(* CODESYS project IndraLogic.project

Project tree, tasks and I/O mapping:
  IndraMotionMlc1 : IndraMotion MLC L25, Bosch Rexroth AG, order no. R911171363, version 14.20.34.0
    application Application
      libraries: VisuDialogs, * (System)
      task PlcTask (cyclic, interval 25 ms, priority 5, watchdog 100 ms x 2) calls prgVisualization, prgDataSimulator, PrgBedinpult_Visu
      global variables UserVarGlobal
      Symbols
      global variables MlcVarGlobal
      image pool ImagePool
      Funktionsbausteine/
        function block GenAngleTest [ST]
        function block GenNumTest [ST]
        function block TestGen [FBD]
        function block Tweener [SFC]: SetResToStart, IncResult, DecResult, SetResultToFinal
      Programme/
        program prgVisualization [ST]
        program prgDataSimulator [ST]
      Structs/
        data type TestStruct
      Bedinpult_Visu/
        program PrgBedinpult_Visu [LD]
      HMI/
        visualisation viAttitudeIndicator
      Frames/
        visualisation frBedinpult
        visualisation frSelfTestLamp
    Inline_I_O : Inline I/O, Bosch Rexroth AG, version 12.8.2.0
    Sercos_III_Master : SercosIII Master, Rexroth, order no. 1, version 14.6.0.0
  text list GlobalTextList
  5ce3da45-db07-42e7-a21c-a00fff4ed8f6|C:\Users\Kun\Desktop\Uni\Automatisierungstechnik\ProjektaufgabeAT\Overlay.png
  5ce3da45-db07-42e7-a21c-a00fff4ed8f6|C:\Users\Ghaith\Desktop\Modellfabrik\Logo.jpg
*)

// IndraMotionMlc1/Application/Structs/TestStruct
TYPE TestStruct :
STRUCT
	bEnable		: BOOL;
	iStartValue	: INT;
	iFinalValue	: INT;
	rSweepInc	: REAL;
	bTestActive	: BOOL;
END_STRUCT
END_TYPE

// IndraMotionMlc1/Application/UserVarGlobal
{attribute 'qualified_only'}
VAR_GLOBAL
	bSelfTestAtStartup : BOOL	:= TRUE;
	
	rPitch 		: 	REAL;
	rRoll 		: 	REAL;
	iHeight		:	INT;
	uiSpeed		:	UINT;
	
	rPitch_Input 		: 	REAL;
	rRoll_Input 		: 	REAL;
	iHeight_Input		:	INT;
	uiSpeed_Input		:	UINT;
	
	bAutomatic_Mode_Input	: BOOL;
END_VAR

// IndraMotionMlc1/Application/MlcVarGlobal
(* Automatically generated code by XLC/MLC. *)
(* Please don't edit, the code will be overwritten. For usercode use UserVarGlobal! *)
{attribute 'linkalways'}
{attribute 'analysis' := '-33'}
VAR_GLOBAL CONSTANT

(*Probe 001*)
TouchProbe001: TOUCHPROBE_REF :=(CntrlNo:=LOCAL_CNTRL,TouchProbeNo:=TOUCHPROBE_1);

(*Probe 002*)
TouchProbe002: TOUCHPROBE_REF :=(CntrlNo:=LOCAL_CNTRL,TouchProbeNo:=TOUCHPROBE_2);

(*Probe 003*)
TouchProbe003: TOUCHPROBE_REF :=(CntrlNo:=LOCAL_CNTRL,TouchProbeNo:=TOUCHPROBE_3);

(*Probe 004*)
TouchProbe004: TOUCHPROBE_REF :=(CntrlNo:=LOCAL_CNTRL,TouchProbeNo:=TOUCHPROBE_4);

(*Probe 005*)
TouchProbe005: TOUCHPROBE_REF :=(CntrlNo:=LOCAL_CNTRL,TouchProbeNo:=TOUCHPROBE_5);

(*Probe 006*)
TouchProbe006: TOUCHPROBE_REF :=(CntrlNo:=LOCAL_CNTRL,TouchProbeNo:=TOUCHPROBE_6);

(*Probe 007*)
TouchProbe007: TOUCHPROBE_REF :=(CntrlNo:=LOCAL_CNTRL,TouchProbeNo:=TOUCHPROBE_7);

(*Probe 008*)
TouchProbe008: TOUCHPROBE_REF :=(CntrlNo:=LOCAL_CNTRL,TouchProbeNo:=TOUCHPROBE_8);

(*Probe 009*)
TouchProbe009: TOUCHPROBE_REF :=(CntrlNo:=LOCAL_CNTRL,TouchProbeNo:=TOUCHPROBE_9);

(*Probe 010*)
TouchProbe010: TOUCHPROBE_REF :=(CntrlNo:=LOCAL_CNTRL,TouchProbeNo:=TOUCHPROBE_10);

(*Probe 011*)
TouchProbe011: TOUCHPROBE_REF :=(CntrlNo:=LOCAL_CNTRL,TouchProbeNo:=TOUCHPROBE_11);

(*Probe 012*)
TouchProbe012: TOUCHPROBE_REF :=(CntrlNo:=LOCAL_CNTRL,TouchProbeNo:=TOUCHPROBE_12);

(*Probe 013*)
TouchProbe013: TOUCHPROBE_REF :=(CntrlNo:=LOCAL_CNTRL,TouchProbeNo:=TOUCHPROBE_13);

(*Probe 014*)
TouchProbe014: TOUCHPROBE_REF :=(CntrlNo:=LOCAL_CNTRL,TouchProbeNo:=TOUCHPROBE_14);

(*Probe 015*)
TouchProbe015: TOUCHPROBE_REF :=(CntrlNo:=LOCAL_CNTRL,TouchProbeNo:=TOUCHPROBE_15);

(*Probe 016*)
TouchProbe016: TOUCHPROBE_REF :=(CntrlNo:=LOCAL_CNTRL,TouchProbeNo:=TOUCHPROBE_16);

(*Probe 017*)
TouchProbe017: TOUCHPROBE_REF :=(CntrlNo:=LOCAL_CNTRL,TouchProbeNo:=TOUCHPROBE_17);

(*Probe 018*)
TouchProbe018: TOUCHPROBE_REF :=(CntrlNo:=LOCAL_CNTRL,TouchProbeNo:=TOUCHPROBE_18);

(*Probe 019*)
TouchProbe019: TOUCHPROBE_REF :=(CntrlNo:=LOCAL_CNTRL,TouchProbeNo:=TOUCHPROBE_19);

(*Probe 020*)
TouchProbe020: TOUCHPROBE_REF :=(CntrlNo:=LOCAL_CNTRL,TouchProbeNo:=TOUCHPROBE_20);

(*Probe 021*)
TouchProbe021: TOUCHPROBE_REF :=(CntrlNo:=LOCAL_CNTRL,TouchProbeNo:=TOUCHPROBE_21);

(*Probe 022*)
TouchProbe022: TOUCHPROBE_REF :=(CntrlNo:=LOCAL_CNTRL,TouchProbeNo:=TOUCHPROBE_22);

(*Probe 023*)
TouchProbe023: TOUCHPROBE_REF :=(CntrlNo:=LOCAL_CNTRL,TouchProbeNo:=TOUCHPROBE_23);

(*Probe 024*)
TouchProbe024: TOUCHPROBE_REF :=(CntrlNo:=LOCAL_CNTRL,TouchProbeNo:=TOUCHPROBE_24);

(*Probe 025*)
TouchProbe025: TOUCHPROBE_REF :=(CntrlNo:=LOCAL_CNTRL,TouchProbeNo:=TOUCHPROBE_25);

(*Probe 026*)
TouchProbe026: TOUCHPROBE_REF :=(CntrlNo:=LOCAL_CNTRL,TouchProbeNo:=TOUCHPROBE_26);

(*Probe 027*)
TouchProbe027: TOUCHPROBE_REF :=(CntrlNo:=LOCAL_CNTRL,TouchProbeNo:=TOUCHPROBE_27);

(*Probe 028*)
TouchProbe028: TOUCHPROBE_REF :=(CntrlNo:=LOCAL_CNTRL,TouchProbeNo:=TOUCHPROBE_28);

(*Probe 029*)
TouchProbe029: TOUCHPROBE_REF :=(CntrlNo:=LOCAL_CNTRL,TouchProbeNo:=TOUCHPROBE_29);

(*Probe 030*)
TouchProbe030: TOUCHPROBE_REF :=(CntrlNo:=LOCAL_CNTRL,TouchProbeNo:=TOUCHPROBE_30);

(*Probe 031*)
TouchProbe031: TOUCHPROBE_REF :=(CntrlNo:=LOCAL_CNTRL,TouchProbeNo:=TOUCHPROBE_31);

(*Probe 032*)
TouchProbe032: TOUCHPROBE_REF :=(CntrlNo:=LOCAL_CNTRL,TouchProbeNo:=TOUCHPROBE_32);

(*Probe 033*)
TouchProbe033: TOUCHPROBE_REF :=(CntrlNo:=LOCAL_CNTRL,TouchProbeNo:=TOUCHPROBE_33);

(*Probe 034*)
TouchProbe034: TOUCHPROBE_REF :=(CntrlNo:=LOCAL_CNTRL,TouchProbeNo:=TOUCHPROBE_34);

(*Probe 035*)
TouchProbe035: TOUCHPROBE_REF :=(CntrlNo:=LOCAL_CNTRL,TouchProbeNo:=TOUCHPROBE_35);

(*Probe 036*)
TouchProbe036: TOUCHPROBE_REF :=(CntrlNo:=LOCAL_CNTRL,TouchProbeNo:=TOUCHPROBE_36);

(*Probe 037*)
TouchProbe037: TOUCHPROBE_REF :=(CntrlNo:=LOCAL_CNTRL,TouchProbeNo:=TOUCHPROBE_37);

(*Probe 038*)
TouchProbe038: TOUCHPROBE_REF :=(CntrlNo:=LOCAL_CNTRL,TouchProbeNo:=TOUCHPROBE_38);

(*Probe 039*)
TouchProbe039: TOUCHPROBE_REF :=(CntrlNo:=LOCAL_CNTRL,TouchProbeNo:=TOUCHPROBE_39);

(*Probe 040*)
TouchProbe040: TOUCHPROBE_REF :=(CntrlNo:=LOCAL_CNTRL,TouchProbeNo:=TOUCHPROBE_40);

(*Probe 041*)
TouchProbe041: TOUCHPROBE_REF :=(CntrlNo:=LOCAL_CNTRL,TouchProbeNo:=TOUCHPROBE_41);

(*Probe 042*)
TouchProbe042: TOUCHPROBE_REF :=(CntrlNo:=LOCAL_CNTRL,TouchProbeNo:=TOUCHPROBE_42);

(*Probe 043*)
TouchProbe043: TOUCHPROBE_REF :=(CntrlNo:=LOCAL_CNTRL,TouchProbeNo:=TOUCHPROBE_43);

(*Probe 044*)
TouchProbe044: TOUCHPROBE_REF :=(CntrlNo:=LOCAL_CNTRL,TouchProbeNo:=TOUCHPROBE_44);

(*Probe 045*)
TouchProbe045: TOUCHPROBE_REF :=(CntrlNo:=LOCAL_CNTRL,TouchProbeNo:=TOUCHPROBE_45);

(*Probe 046*)
TouchProbe046: TOUCHPROBE_REF :=(CntrlNo:=LOCAL_CNTRL,TouchProbeNo:=TOUCHPROBE_46);

(*Probe 047*)
TouchProbe047: TOUCHPROBE_REF :=(CntrlNo:=LOCAL_CNTRL,TouchProbeNo:=TOUCHPROBE_47);

(*Probe 048*)
TouchProbe048: TOUCHPROBE_REF :=(CntrlNo:=LOCAL_CNTRL,TouchProbeNo:=TOUCHPROBE_48);

(*Probe 049*)
TouchProbe049: TOUCHPROBE_REF :=(CntrlNo:=LOCAL_CNTRL,TouchProbeNo:=TOUCHPROBE_49);

(*Probe 050*)
TouchProbe050: TOUCHPROBE_REF :=(CntrlNo:=LOCAL_CNTRL,TouchProbeNo:=TOUCHPROBE_50);

(*Probe 051*)
TouchProbe051: TOUCHPROBE_REF :=(CntrlNo:=LOCAL_CNTRL,TouchProbeNo:=TOUCHPROBE_51);

(*Probe 052*)
TouchProbe052: TOUCHPROBE_REF :=(CntrlNo:=LOCAL_CNTRL,TouchProbeNo:=TOUCHPROBE_52);

(*Probe 053*)
TouchProbe053: TOUCHPROBE_REF :=(CntrlNo:=LOCAL_CNTRL,TouchProbeNo:=TOUCHPROBE_53);

(*Probe 054*)
TouchProbe054: TOUCHPROBE_REF :=(CntrlNo:=LOCAL_CNTRL,TouchProbeNo:=TOUCHPROBE_54);

(*Probe 055*)
TouchProbe055: TOUCHPROBE_REF :=(CntrlNo:=LOCAL_CNTRL,TouchProbeNo:=TOUCHPROBE_55);

(*Probe 056*)
TouchProbe056: TOUCHPROBE_REF :=(CntrlNo:=LOCAL_CNTRL,TouchProbeNo:=TOUCHPROBE_56);

(*Probe 057*)
TouchProbe057: TOUCHPROBE_REF :=(CntrlNo:=LOCAL_CNTRL,TouchProbeNo:=TOUCHPROBE_57);

(*Probe 058*)
TouchProbe058: TOUCHPROBE_REF :=(CntrlNo:=LOCAL_CNTRL,TouchProbeNo:=TOUCHPROBE_58);

(*Probe 059*)
TouchProbe059: TOUCHPROBE_REF :=(CntrlNo:=LOCAL_CNTRL,TouchProbeNo:=TOUCHPROBE_59);

(*Probe 060*)
TouchProbe060: TOUCHPROBE_REF :=(CntrlNo:=LOCAL_CNTRL,TouchProbeNo:=TOUCHPROBE_60);

(*Probe 061*)
TouchProbe061: TOUCHPROBE_REF :=(CntrlNo:=LOCAL_CNTRL,TouchProbeNo:=TOUCHPROBE_61);

(*Probe 062*)
TouchProbe062: TOUCHPROBE_REF :=(CntrlNo:=LOCAL_CNTRL,TouchProbeNo:=TOUCHPROBE_62);

(*Probe 063*)
TouchProbe063: TOUCHPROBE_REF :=(CntrlNo:=LOCAL_CNTRL,TouchProbeNo:=TOUCHPROBE_63);

(*Probe 064*)
TouchProbe064: TOUCHPROBE_REF :=(CntrlNo:=LOCAL_CNTRL,TouchProbeNo:=TOUCHPROBE_64);

(*Probe 065*)
TouchProbe065: TOUCHPROBE_REF :=(CntrlNo:=LOCAL_CNTRL,TouchProbeNo:=TOUCHPROBE_65);

(*Probe 066*)
TouchProbe066: TOUCHPROBE_REF :=(CntrlNo:=LOCAL_CNTRL,TouchProbeNo:=TOUCHPROBE_66);

(*Probe 067*)
TouchProbe067: TOUCHPROBE_REF :=(CntrlNo:=LOCAL_CNTRL,TouchProbeNo:=TOUCHPROBE_67);

(*Probe 068*)
TouchProbe068: TOUCHPROBE_REF :=(CntrlNo:=LOCAL_CNTRL,TouchProbeNo:=TOUCHPROBE_68);

(*Probe 069*)
TouchProbe069: TOUCHPROBE_REF :=(CntrlNo:=LOCAL_CNTRL,TouchProbeNo:=TOUCHPROBE_69);

(*Probe 070*)
TouchProbe070: TOUCHPROBE_REF :=(CntrlNo:=LOCAL_CNTRL,TouchProbeNo:=TOUCHPROBE_70);

(*Probe 071*)
TouchProbe071: TOUCHPROBE_REF :=(CntrlNo:=LOCAL_CNTRL,TouchProbeNo:=TOUCHPROBE_71);

(*Probe 072*)
TouchProbe072: TOUCHPROBE_REF :=(CntrlNo:=LOCAL_CNTRL,TouchProbeNo:=TOUCHPROBE_72);

(*Probe 073*)
TouchProbe073: TOUCHPROBE_REF :=(CntrlNo:=LOCAL_CNTRL,TouchProbeNo:=TOUCHPROBE_73);

(*Probe 074*)
TouchProbe074: TOUCHPROBE_REF :=(CntrlNo:=LOCAL_CNTRL,TouchProbeNo:=TOUCHPROBE_74);

(*Probe 075*)
TouchProbe075: TOUCHPROBE_REF :=(CntrlNo:=LOCAL_CNTRL,TouchProbeNo:=TOUCHPROBE_75);

(*Probe 076*)
TouchProbe076: TOUCHPROBE_REF :=(CntrlNo:=LOCAL_CNTRL,TouchProbeNo:=TOUCHPROBE_76);

(*Probe 077*)
TouchProbe077: TOUCHPROBE_REF :=(CntrlNo:=LOCAL_CNTRL,TouchProbeNo:=TOUCHPROBE_77);

(*Probe 078*)
TouchProbe078: TOUCHPROBE_REF :=(CntrlNo:=LOCAL_CNTRL,TouchProbeNo:=TOUCHPROBE_78);

(*Probe 079*)
TouchProbe079: TOUCHPROBE_REF :=(CntrlNo:=LOCAL_CNTRL,TouchProbeNo:=TOUCHPROBE_79);

(*Probe 080*)
TouchProbe080: TOUCHPROBE_REF :=(CntrlNo:=LOCAL_CNTRL,TouchProbeNo:=TOUCHPROBE_80);

(*Probe 081*)
TouchProbe081: TOUCHPROBE_REF :=(CntrlNo:=LOCAL_CNTRL,TouchProbeNo:=TOUCHPROBE_81);

(*Probe 082*)
TouchProbe082: TOUCHPROBE_REF :=(CntrlNo:=LOCAL_CNTRL,TouchProbeNo:=TOUCHPROBE_82);

(*Probe 083*)
TouchProbe083: TOUCHPROBE_REF :=(CntrlNo:=LOCAL_CNTRL,TouchProbeNo:=TOUCHPROBE_83);

(*Probe 084*)
TouchProbe084: TOUCHPROBE_REF :=(CntrlNo:=LOCAL_CNTRL,TouchProbeNo:=TOUCHPROBE_84);

(*Probe 085*)
TouchProbe085: TOUCHPROBE_REF :=(CntrlNo:=LOCAL_CNTRL,TouchProbeNo:=TOUCHPROBE_85);

(*Probe 086*)
TouchProbe086: TOUCHPROBE_REF :=(CntrlNo:=LOCAL_CNTRL,TouchProbeNo:=TOUCHPROBE_86);

(*Probe 087*)
TouchProbe087: TOUCHPROBE_REF :=(CntrlNo:=LOCAL_CNTRL,TouchProbeNo:=TOUCHPROBE_87);

(*Probe 088*)
TouchProbe088: TOUCHPROBE_REF :=(CntrlNo:=LOCAL_CNTRL,TouchProbeNo:=TOUCHPROBE_88);

(*Probe 089*)
TouchProbe089: TOUCHPROBE_REF :=(CntrlNo:=LOCAL_CNTRL,TouchProbeNo:=TOUCHPROBE_89);

(*Probe 090*)
TouchProbe090: TOUCHPROBE_REF :=(CntrlNo:=LOCAL_CNTRL,TouchProbeNo:=TOUCHPROBE_90);

(*Probe 091*)
TouchProbe091: TOUCHPROBE_REF :=(CntrlNo:=LOCAL_CNTRL,TouchProbeNo:=TOUCHPROBE_91);

(*Probe 092*)
TouchProbe092: TOUCHPROBE_REF :=(CntrlNo:=LOCAL_CNTRL,TouchProbeNo:=TOUCHPROBE_92);

(*Probe 093*)
TouchProbe093: TOUCHPROBE_REF :=(CntrlNo:=LOCAL_CNTRL,TouchProbeNo:=TOUCHPROBE_93);

(*Probe 094*)
TouchProbe094: TOUCHPROBE_REF :=(CntrlNo:=LOCAL_CNTRL,TouchProbeNo:=TOUCHPROBE_94);

(*Probe 095*)
TouchProbe095: TOUCHPROBE_REF :=(CntrlNo:=LOCAL_CNTRL,TouchProbeNo:=TOUCHPROBE_95);

(*Probe 096*)
TouchProbe096: TOUCHPROBE_REF :=(CntrlNo:=LOCAL_CNTRL,TouchProbeNo:=TOUCHPROBE_96);

(*Probe 097*)
TouchProbe097: TOUCHPROBE_REF :=(CntrlNo:=LOCAL_CNTRL,TouchProbeNo:=TOUCHPROBE_97);

(*Probe 098*)
TouchProbe098: TOUCHPROBE_REF :=(CntrlNo:=LOCAL_CNTRL,TouchProbeNo:=TOUCHPROBE_98);

(*Probe 099*)
TouchProbe099: TOUCHPROBE_REF :=(CntrlNo:=LOCAL_CNTRL,TouchProbeNo:=TOUCHPROBE_99);

(*Probe 100*)
TouchProbe100: TOUCHPROBE_REF :=(CntrlNo:=LOCAL_CNTRL,TouchProbeNo:=TOUCHPROBE_100);

END_VAR

// IndraMotionMlc1/Application/Programme/prgVisualization
PROGRAM prgVisualization
VAR
	rPitch_Visu 	: 	REAL;
	rRoll_Visu		: 	REAL;
	iHeight_Visu		:	INT;
	uiSpeed_Visu		:	UINT;
	bDisableControlPanel: BOOL;
END_VAR

VAR CONSTANT
	
END_VAR

rRoll_Visu := UserVarGlobal.rRoll;
iHeight_Visu := UserVarGlobal.iHeight;
rPitch_Visu := UserVarGlobal.rPitch * 4;
uiSpeed_Visu :=UserVarGlobal.uiSpeed;

IF ((UserVarGlobal.bAutomatic_Mode_Input = FALSE AND (rRoll_Visu <> UserVarGlobal.rRoll_Input OR rPitch_Visu <> UserVarGlobal.rPitch_Input*4 OR iHeight_Visu <> UserVarGlobal.iHeight_Input OR uiSpeed_Visu <> UserVarGlobal.uiSpeed_Input)) OR UserVarGlobal.bSelfTestAtStartup) THEN
	bDisableControlPanel := TRUE;
ELSE
	bDisableControlPanel := FALSE;
END_IF

END_PROGRAM

// IndraMotionMlc1/Application/Programme/prgDataSimulator
PROGRAM prgDataSimulator
VAR
	rPitch 			: 	REAL;
	rRoll 			: 	REAL;
	iHeight			:	INT;
	uiSpeed			:	UINT;
	
	// Internal Variables for Automatic Operation
	fbTestGenerator		:	TestGen;
	suPitchTestStruct	:	testStruct;
	suRollTestStruct	:	testStruct;
	suHeightTestStruct  :	testStruct;
	suSpeedTestStruct	:	testStruct;
	bInit				:	BOOL := TRUE;
	
	// Internal Variables for Manual Operation
	fbPitchTween		: Tweener;
	fbRollTween			: Tweener;
	fbHeightTween		: Tweener;
	fbSpeedTween		: Tweener;
	
	siSweepInc		:	SINT	:=	1;
END_VAR

// Initialize Test Structs
IF bInit THEN
	suRollTestStruct.bEnable 		:= TRUE;
	suRollTestStruct.iStartValue 	:= -30;
	suRollTestStruct.iFinalValue 	:= 30;
	suRollTestStruct.rSweepInc 	:= 0.6;
	
	suHeightTestStruct.bEnable 	:= TRUE;
	suHeightTestStruct.iStartValue	:= 0;
	suHeightTestStruct.iFinalValue := 1000;
	suHeightTestStruct.rSweepInc	:= 30;
	
	suPitchTestStruct.bEnable 	:= TRUE;
	suPitchTestStruct.iStartValue	:= 20;
	suPitchTestStruct.iFinalValue 	:= -20;
	suPitchTestStruct.rSweepInc	:= 0.8;
	
	suSpeedTestStruct.bEnable 	:= TRUE;
	suSpeedTestStruct.iStartValue	:= 0;
	suSpeedTestStruct.iFinalValue 	:= 500;
	suSpeedTestStruct.rSweepInc	:= 15;
	
	bInit := FALSE;
END_IF

// Run Self Test at Startup
IF (UserVarGlobal.bSelfTestAtStartup OR UserVarGlobal.bAutomatic_Mode_Input) THEN
		
	fbTestGenerator(suPitchTestStruct:=suPitchTestStruct,suRollTestStruct:=suRollTestStruct , suHeightTestStruct:=suHeightTestStruct, suSpeedTestStruct:=suSpeedTestStruct);
	
	suPitchTestStruct.bEnable := TRUE;
	suRollTestStruct.bEnable := TRUE;
	suHeightTestStruct.bEnable := TRUE;
	suSpeedTestStruct.bEnable := TRUE;
	
	rPitch := fbTestGenerator.rPitch;
	rRoll := fbTestGenerator.rRoll;
	iHeight := fbTestGenerator.iHeight;
	uiSpeed := fbTestGenerator.uiSpeed;
	IF (NOT fbTestGenerator.bTestActive) THEN
		// When no all Tests are done, set all Variables to 0
		rPitch := 0;
		rRoll := 0;
		iHeight := 0;
		uiSpeed := 0;
		suPitchTestStruct.bEnable := FALSE;
		suRollTestStruct.bEnable := FALSE;
		suHeightTestStruct.bEnable := FALSE;
		suSpeedTestStruct.bEnable := FALSE;
		UserVarGlobal.bSelfTestAtStartup := FALSE;
	END_IF
ELSIF (UserVarGlobal.bAutomatic_Mode_Input = FALSE) THEN
	suPitchTestStruct.bEnable := FALSE;
	suRollTestStruct.bEnable := FALSE;
	suHeightTestStruct.bEnable := FALSE;
	suSpeedTestStruct.bEnable := FALSE;
	// Animate between current point and input
	fbPitchTween(rStartNum:=rPitch,rFinalNum:=UserVarGlobal.rPitch_Input,rIncrement:=siSweepInc);
	rPitch := fbPitchTween.rResult;
	fbRollTween(rStartNum:=rRoll,rFinalNum:=UserVarGlobal.rRoll_Input,rIncrement:=siSweepInc);
	rRoll := fbRollTween.rResult;
	fbHeightTween(rStartNum:=iHeight,rFinalNum:=UserVarGlobal.iHeight_Input,rIncrement:=siSweepInc*5);
	iHeight := fbHeightTween.iResult;
	fbSpeedTween(rStartNum:=uiSpeed,rFinalNum:=UserVarGlobal.uiSpeed_Input,rIncrement:=siSweepInc*5);
	uiSpeed := fbSpeedTween.iResult;
END_IF 

UserVarGlobal.rPitch := rPitch;
UserVarGlobal.rRoll := rRoll;
UserVarGlobal.iHeight := iHeight;
UserVarGlobal.uiSpeed := uiSpeed;

END_PROGRAM

// IndraMotionMlc1/Application/Funktionsbausteine/TestGen
FUNCTION_BLOCK TestGen
VAR_INPUT
	suPitchTestStruct		: TestStruct;
	suRollTestStruct		: TestStruct;
	suHeightTestStruct	: TestStruct;
	suSpeedTestStruct		: TestStruct;
END_VAR
VAR_OUTPUT
	rPitch			: REAL;
	rRoll			: REAL;
	iHeight			: INT;
	uiSpeed			: UINT;
	bTestActive		: BOOL;
END_VAR
VAR
	fbPitchTest		: GenAngleTest;
	fbRollTest		: GenAngleTest;
	fbHeightTest		: GenNumTest;
	fbSpeedTest		: GenNumTest;
	
	// Einschaltverzoegerung zwischen Tests
	tiTon_Time		: TIME := T#0.5S;
	tiTon_Et		: TIME;
	TON_roll		: TON;
	TON_height		: TON;
	TON_speed		: TON;

END_VAR

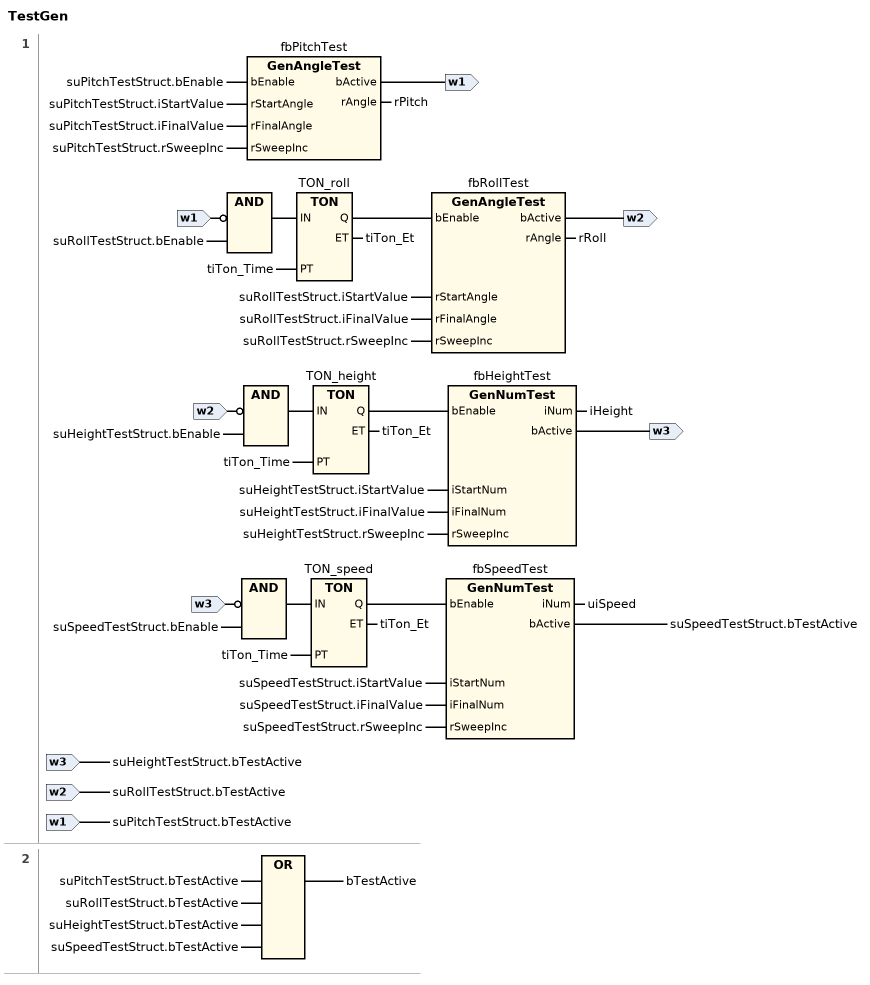
// NETWORK 1
fbPitchTest(
    bEnable := suPitchTestStruct.bEnable,
    rStartAngle := suPitchTestStruct.iStartValue,
    rFinalAngle := suPitchTestStruct.iFinalValue,
    rSweepInc := suPitchTestStruct.rSweepInc,
    rAngle => rPitch); // GenAngleTest
TON_roll(IN := NOT fbPitchTest.bActive AND suRollTestStruct.bEnable, PT := tiTon_Time, ET => tiTon_Et); // TON
fbRollTest(
    bEnable := TON_roll.Q,
    rStartAngle := suRollTestStruct.iStartValue,
    rFinalAngle := suRollTestStruct.iFinalValue,
    rSweepInc := suRollTestStruct.rSweepInc,
    rAngle => rRoll); // GenAngleTest
TON_height(IN := NOT fbRollTest.bActive AND suHeightTestStruct.bEnable, PT := tiTon_Time, ET => tiTon_Et); // TON
fbHeightTest(
    bEnable := TON_height.Q,
    iStartNum := suHeightTestStruct.iStartValue,
    iFinalNum := suHeightTestStruct.iFinalValue,
    rSweepInc := suHeightTestStruct.rSweepInc,
    iNum => iHeight); // GenNumTest
TON_speed(IN := NOT fbHeightTest.bActive AND suSpeedTestStruct.bEnable, PT := tiTon_Time, ET => tiTon_Et); // TON
fbSpeedTest(
    bEnable := TON_speed.Q,
    iStartNum := suSpeedTestStruct.iStartValue,
    iFinalNum := suSpeedTestStruct.iFinalValue,
    rSweepInc := suSpeedTestStruct.rSweepInc,
    iNum => uiSpeed); // GenNumTest
suSpeedTestStruct.bTestActive := fbSpeedTest.bActive;
suHeightTestStruct.bTestActive := fbHeightTest.bActive;
suRollTestStruct.bTestActive := fbRollTest.bActive;
suPitchTestStruct.bTestActive := fbPitchTest.bActive;

// NETWORK 2
bTestActive := suPitchTestStruct.bTestActive OR suRollTestStruct.bTestActive OR suHeightTestStruct.bTestActive OR suSpeedTestStruct.bTestActive;

END_FUNCTION_BLOCK

// IndraMotionMlc1/Application/Funktionsbausteine/GenAngleTest
FUNCTION_BLOCK GenAngleTest
VAR_INPUT
	bEnable			: BOOL;
	rStartAngle		: REAL;
	rFinalAngle		: REAL;
	rSweepInc		: REAL;	// Value by which the result is incremented by cycle
END_VAR
VAR_OUTPUT
	bActive			: BOOL := TRUE;
	rAngle			: REAL;
END_VAR
VAR
	bFirstSweep		: BOOL := TRUE;	// Winkel soll einmal in beide Richtugnen verändert werden
	fbTween			: Tweener;
END_VAR

IF (bEnable AND bFirstSweep AND bActive) THEN
	fbTween(rStartNum:=rStartAngle,rFinalNum:=rFinalAngle,rIncrement:=rSweepInc);
	rAngle := fbTween.rResult;
	IF (rAngle = rFinalAngle) THEN
		bFirstSweep := FALSE;
	END_IF
ELSIF (bEnable AND bFirstSweep = FALSE AND bActive) THEN
	fbTween(rStartNum:=rFinalAngle,rFinalNum:=rStartAngle,rIncrement:=rSweepInc);
	rAngle := fbTween.rResult;
	IF (rAngle = rStartAngle AND fbTween.bActive = FALSE) THEN
		bActive := FALSE;
		bFirstSweep := TRUE;
		rAngle := 0;
	END_IF
END_IF

IF (bEnable = FALSE) THEN
	rAngle := 0;
	bFirstSweep := TRUE;
	bActive := TRUE;
END_IF

END_FUNCTION_BLOCK

// IndraMotionMlc1/Application/Funktionsbausteine/Tweener
FUNCTION_BLOCK Tweener
VAR_INPUT
	rStartNum	:	REAL;
	rFinalNum	:	REAL;
	rIncrement	:	REAL;
END_VAR
VAR_OUTPUT
	rResult			:	REAL;
	iResult			:	INT;
	bActive			:	BOOL;
END_VAR

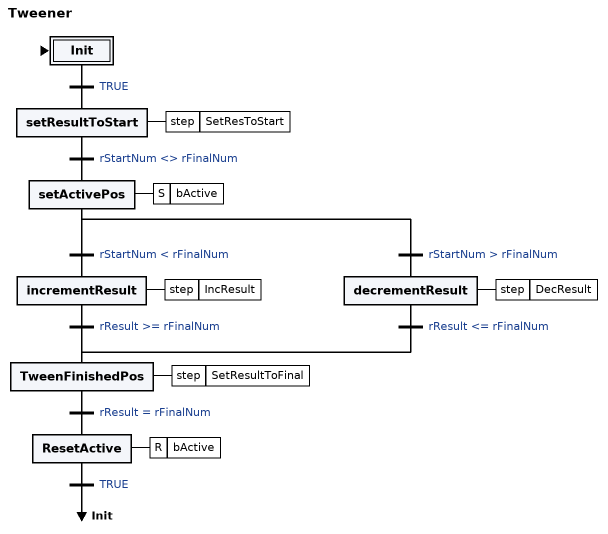
INITIAL_STEP Init:
END_STEP
TRANSITION FROM Init TO setResultToStart
    := TRUE;
END_TRANSITION
STEP setResultToStart:
    SetResToStart(N);  // step action
END_STEP
TRANSITION FROM setResultToStart TO setActivePos
    := rStartNum <> rFinalNum;
END_TRANSITION
STEP setActivePos:
    bActive(S);
END_STEP
TRANSITION FROM setActivePos TO incrementResult
    := rStartNum < rFinalNum;
END_TRANSITION
STEP incrementResult:
    IncResult(N);  // step action
END_STEP
TRANSITION FROM incrementResult TO TweenFinishedPos
    := rResult >= rFinalNum;
END_TRANSITION
TRANSITION FROM setActivePos TO decrementResult
    := rStartNum > rFinalNum;
END_TRANSITION
STEP decrementResult:
    DecResult(N);  // step action
END_STEP
TRANSITION FROM decrementResult TO TweenFinishedPos
    := rResult <= rFinalNum;
END_TRANSITION
STEP TweenFinishedPos:
    SetResultToFinal(N);  // step action
END_STEP
TRANSITION FROM TweenFinishedPos TO ResetActive
    := rResult = rFinalNum;
END_TRANSITION
STEP ResetActive:
    bActive(R);
END_STEP
TRANSITION FROM ResetActive TO Init
    := TRUE;
END_TRANSITION

ACTION SetResToStart:
rResult := rStartNum;
END_ACTION

ACTION IncResult:
rResult := rResult + rIncrement;
iResult := TRUNC_INT(rResult);
END_ACTION

ACTION DecResult:
rResult := rResult - rIncrement;
iResult := TRUNC_INT(rResult);
END_ACTION

ACTION SetResultToFinal:
rResult := rFinalNum;
iResult := TRUNC_INT(rFinalNum);
END_ACTION

END_FUNCTION_BLOCK

// IndraMotionMlc1/Application/Funktionsbausteine/GenNumTest
FUNCTION_BLOCK GenNumTest
VAR_INPUT
	bEnable			: BOOL;
	iStartNum		: INT;
	iFinalNum		: INT;
	rSweepInc		: REAL;	// Value by which the result is incremented by cycle
END_VAR
VAR_OUTPUT
	iNum				: INT;
	bActive			: BOOL := TRUE;
END_VAR
VAR
	bFirstSweep		: BOOL	:= TRUE;
	fbTween			: Tweener;
END_VAR

IF (bEnable AND bFirstSweep AND bActive) THEN
	fbTween(rStartNum:=iStartNum,rFinalNum:=iFinalNum,rIncrement:=rSweepInc);
	iNum := fbTween.iResult;
	IF (iNum = iFinalNum) THEN
		bFirstSweep := FALSE;
	END_IF
ELSIF (bEnable AND bFirstSweep = FALSE AND bActive) THEN
	iNum := fbTween.iResult;
	fbTween(rStartNum:=iFinalNum,rFinalNum:=iStartNum,rIncrement:=rSweepInc);	
	IF (iNum = iStartNum AND fbTween.bActive = FALSE) THEN
		bActive := FALSE;
		bFirstSweep := TRUE;
		iNum := 0;
	END_IF
END_IF

IF (bEnable = FALSE) THEN
	iNum := 0;
	bFirstSweep := TRUE;
	bActive := TRUE;
END_IF

END_FUNCTION_BLOCK

// IndraMotionMlc1/Application/Bedinpult_Visu/PrgBedinpult_Visu
PROGRAM PrgBedinpult_Visu
VAR
blampe_Autmatik		  				:BOOL;//Lampe für Autmatikbetrieb
blampe_Manual		  				:BOOL;//Lampe für Handbetrieb
bSchalter_Automatik_Visu		 	: BOOL; // Umschalter Automatik =1 / Handbetrieb =0 
END_VAR
VAR // added by the converter: edge detectors and wires of the graphical bodies
    _w1 : BOOL;
END_VAR

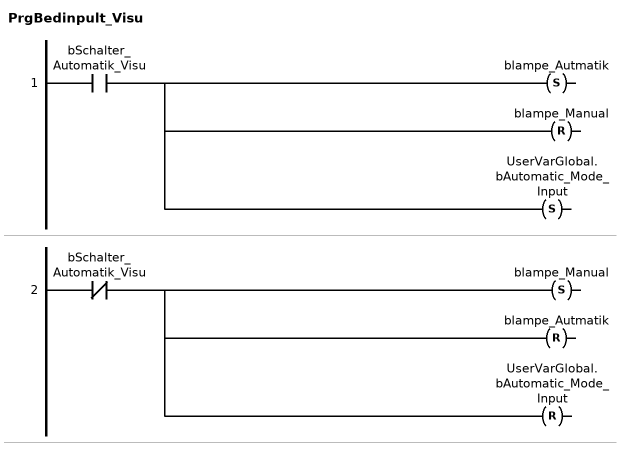
// NETWORK 1
blampe_Autmatik S= bSchalter_Automatik_Visu;
blampe_Manual R= bSchalter_Automatik_Visu;
UserVarGlobal.bAutomatic_Mode_Input S= bSchalter_Automatik_Visu;

// NETWORK 2
_w1 := NOT bSchalter_Automatik_Visu;
blampe_Manual S= _w1;
blampe_Autmatik R= _w1;
UserVarGlobal.bAutomatic_Mode_Input R= _w1;

END_PROGRAM

// IndraMotionMlc1/Application/HMI/viAttitudeIndicator
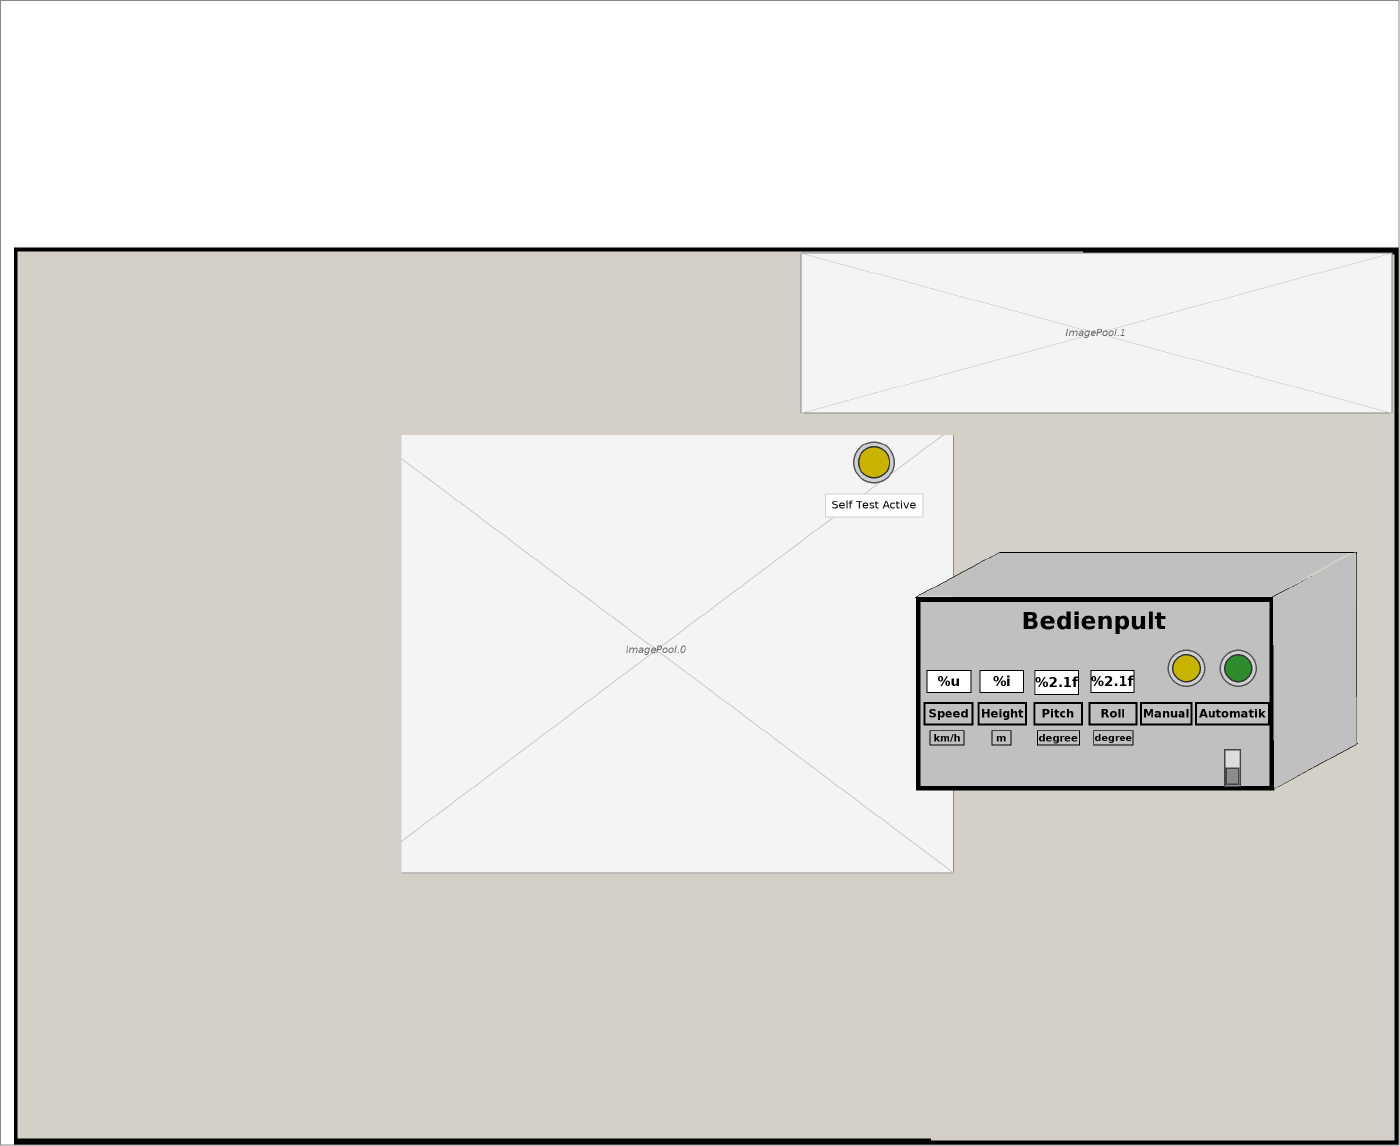
VISUALIZATION viAttitudeIndicator  // 1424x1166
    Rectangle (14,252 1408x912)
    Rectangle (390,660 575x300)
        p2858320360: prgVisualization.rRoll_Visu
        p2773130477: prgVisualization.rPitch_Visu
        p1126004900: prgVisualization.rPitch_Visu
    Rectangle (390,357 575x300)
        p2858320360: prgVisualization.rRoll_Visu
        p2773130477: prgVisualization.rPitch_Visu
        p1126004900: prgVisualization.rPitch_Visu
    Ellipse (515,510 300x300)
    Line (565,660) (765,660)
    Line (640,640) (690,640)
        p2858320360: prgVisualization.rRoll_Visu
        p2773130477: prgVisualization.rPitch_Visu
        p1126004900: prgVisualization.rPitch_Visu
    Line (615,620) (715,620)
        p2858320360: prgVisualization.rRoll_Visu
        p2773130477: prgVisualization.rPitch_Visu
        p1126004900: prgVisualization.rPitch_Visu
    Line (640,600) (690,600)
        p2858320360: prgVisualization.rRoll_Visu
        p2773130477: prgVisualization.rPitch_Visu
        p1126004900: prgVisualization.rPitch_Visu
    Line (640,680) (690,680)
        p2858320360: prgVisualization.rRoll_Visu
        p2773130477: prgVisualization.rPitch_Visu
        p1126004900: prgVisualization.rPitch_Visu
    Line (615,700) (715,700)
        p2858320360: prgVisualization.rRoll_Visu
        p2773130477: prgVisualization.rPitch_Visu
        p1126004900: prgVisualization.rPitch_Visu
    Line (640,720) (690,720)
        p2858320360: prgVisualization.rRoll_Visu
        p2773130477: prgVisualization.rPitch_Visu
        p1126004900: prgVisualization.rPitch_Visu
    Line (615,580) (715,580)
        p2858320360: prgVisualization.rRoll_Visu
        p2773130477: prgVisualization.rPitch_Visu
        p1126004900: prgVisualization.rPitch_Visu
    Line (615,740) (715,740)
        p2858320360: prgVisualization.rRoll_Visu
        p2773130477: prgVisualization.rPitch_Visu
        p1126004900: prgVisualization.rPitch_Visu
    Line (815,660) (790,660)
        p2858320360: prgVisualization.rRoll_Visu
    Line (515,660) (540,660)
        p2858320360: prgVisualization.rRoll_Visu
    Rectangle (715,605 30x28), "10"
        p2858320360: prgVisualization.rRoll_Visu
        p2773130477: prgVisualization.rPitch_Visu
        p1126004900: prgVisualization.rPitch_Visu
    Rectangle (715,565 30x30), "20"
        p2858320360: prgVisualization.rRoll_Visu
        p2773130477: prgVisualization.rPitch_Visu
        p1126004900: prgVisualization.rPitch_Visu
    Rectangle (585,605 30x30), "10"
        p2858320360: prgVisualization.rRoll_Visu
        p2773130477: prgVisualization.rPitch_Visu
        p1126004900: prgVisualization.rPitch_Visu
    Rectangle (585,565 30x30), "20"
        p2858320360: prgVisualization.rRoll_Visu
        p2773130477: prgVisualization.rPitch_Visu
        p1126004900: prgVisualization.rPitch_Visu
    Polyline (655,514) (655,514) (675,514) (665,535) (655,514)
    Rectangle (715,685 30x28), "10"
        p2858320360: prgVisualization.rRoll_Visu
        p2773130477: prgVisualization.rPitch_Visu
        p1126004900: prgVisualization.rPitch_Visu
    Rectangle (585,685 30x28), "10"
        p2858320360: prgVisualization.rRoll_Visu
        p2773130477: prgVisualization.rPitch_Visu
        p1126004900: prgVisualization.rPitch_Visu
    Rectangle (715,725 30x28), "20"
        p2858320360: prgVisualization.rRoll_Visu
        p2773130477: prgVisualization.rPitch_Visu
        p1126004900: prgVisualization.rPitch_Visu
    Rectangle (585,725 30x28), "20"
        p2858320360: prgVisualization.rRoll_Visu
        p2738717112: prgVisualization.rPitch_Visu
    Polyline (654,555) (655,555) (675,555) (665,535) (655,555)
        p2858320360: prgVisualization.rRoll_Visu
    RoundedRectangle (763,631 46x22), "%i", text variable: UserVarGlobal.iHeight, text index: prgVisualization.uiSpeed_Visu
    RoundedRectangle (523,631 46x22), "%u", text variable: UserVarGlobal.uiSpeed
    Line (743,525) (731,547)
    Line (710,538) (719,512)
    Line (688,532) (691,505)
    Line (642,532) (639,509)
    Line (620,538) (612,512)
    Line (600,548) (587,526)
    Rectangle (253,885 876x273)
    Rectangle (947,259 471x901)
    RoundedRectangle (754,589 41x17), "%i", text variable: UserVarGlobal.iHeight_Input, text index: prgVisualization.uiSpeed_Visu
    Image (365,434 605x454), image: ImagePool.0
    Rectangle (18,256 390x902)
    Rectangle (225,256 876x186)
    Image (814,257 602x163), image: ImagePool.1
    Frame (917,547 466x259), input disabled if: prgVisualization.bDisableControlPanel
        shows frBedinpult()
    Frame (839,446 100x100)
        shows frSelfTestLamp(bTestLamp := UserVarGlobal.bSelfTestAtStartup)
END_VISUALIZATION

// IndraMotionMlc1/Application/Frames/frBedinpult
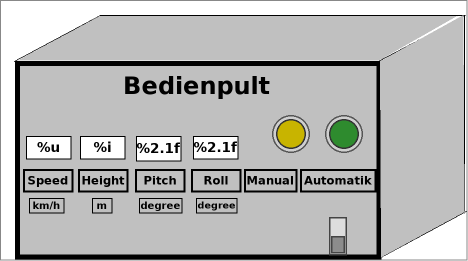
VISUALIZATION frBedinpult  // 468x261
    Rectangle (15,61 366x198)
    Line (14,61) (100,15)
    Polygon (379,60) (458,15) (457,16) (101,15) (18,60)
    Group (23,15 443x243)
        Line (357,181) (355,176)
        DipSwitch (296,199 38x44), variable: PrgBedinpult_Visu.bSchalter_Automatik_Visu, behaviour: TOGGLE, style: Switch-DipSwitch-Gray
        Lamp1 (297,97 48x44), variable: PrgBedinpult_Visu.blampe_Autmatik, style: Lamp-Lamp1-Green
        Lamp1 (246,97 44x44), variable: PrgBedinpult_Visu.blampe_Manual, style: Lamp-Lamp1-Yellow
        Rectangle (277,154 76x23), "Automatik"
        Rectangle (221,154 53x23), "Manual"
        Rectangle (170,121 45x23), "%2.1f", text variable: UserVarGlobal.rRoll_Input
            OnMouseClick: write the text variable via InputWithLimits, min -180, max 179
        Rectangle (0,154 50x23), "Speed"
        Rectangle (112,154 50x23), "Pitch"
        Rectangle (168,154 50x23), "Roll"
        Rectangle (55,154 50x23), "Height"
        Rectangle (113,121 45x25), "%2.1f", text variable: UserVarGlobal.rPitch_Input
            OnMouseClick: write the text variable via InputWithLimits, min -20, max 20
        Rectangle (57,121 45x23), "%i", text variable: UserVarGlobal.iHeight_Input
            OnMouseClick: write the text variable via InputWithLimits, min 0, max 16000
        Rectangle (3,121 45x23), "%u", text variable: UserVarGlobal.uiSpeed_Input
            OnMouseClick: write the text variable via InputWithLimits, min 0, max 2000
        Rectangle (98,59 151x23), "Bedienpult"
        Line (355,46) (442,0)
        Line (356,243) (443,196)
        Line (441,0) (441,198)
        Polygon (354,49) (355,54)
        Line (77,0) (441,0)
        Polygon (357,46) (440,0) (441,198) (442,196) (358,242)
        Rectangle (6,183 35x15), "km/h"
        Rectangle (69,183 20x15), "m"
        Rectangle (116,183 43x15), "degree"
        Rectangle (173,183 41x15), "degree"
END_VISUALIZATION

// IndraMotionMlc1/Application/Frames/frSelfTestLamp
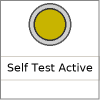
VISUALIZATION frSelfTestLamp  // 100x100
VAR_IN_OUT
	bTestLamp	:	BOOL;
END_VAR
    Lamp1 (25,0 50x49), variable: bTestLamp, style: Lamp-Lamp1-Yellow
    Textfield (0,56 100x24), "Self Test Active", colour toggle: bTestLamp
END_VISUALIZATION
